# EPICS substitutions: beckhoffApp/Db/units_tc.substitutions
file "$(TOP)/beckhoffApp/beckhoff_read_pv.template" {
    pattern {P, NAME, PORT, ADSPORT, V, RECTYPE, EPICSDTYP, ADS_TYPE}
    {"\$(P)", "ASTAXES_\$(AXIS_NUM):STDESC-SUNITS", "\$(PORT)", "\$(ADSPORT)", "GVL.astAxes[\$(AXIS_NUM)].stDescription.sUnits", stringin, "asynOctetRead", "STRING N=32"}
}
